Staubli VAL3: POLYGON.dtx

public num distance
public num moveType = 1
public num nIndexGun
public num nStop
public num nTcpAction = 1
public num nTime
public num nEdge
public num nRotationangle
public num nWidth
public num nLaserDelay = 0.8
public num nLaserPower = 60
public num nGasPressure = 90
public num nFrameIndex
public num nPWMPercent = 100
public num nJointMode
public string comment = "Polygon..."
public string instruction
public bool bCutting
public bool toStop
public bool bRes
public frame fTrack = {fatherId=world[0]}
public jointRx jReadyInOut
public jointRx jConfig
public pointRx pMoveTo = {fatherId=fTrack[0]}
public pointRx pCutting[21]
  [0] = {fatherId=fTrack[0]}
  [1] = {fatherId=fTrack[0]}
  [2] = {fatherId=fTrack[0]}
  [3] = {fatherId=fTrack[0]}
  [4] = {fatherId=fTrack[0]}
  [5] = {fatherId=fTrack[0]}
  [6] = {fatherId=fTrack[0]}
  [7] = {fatherId=fTrack[0]}
  [8] = {fatherId=fTrack[0]}
  [9] = {fatherId=fTrack[0]}
  [10] = {fatherId=fTrack[0]}
  [11] = {fatherId=fTrack[0]}
  [12] = {fatherId=fTrack[0]}
  [13] = {fatherId=fTrack[0]}
  [14] = {fatherId=fTrack[0]}
  [15] = {fatherId=fTrack[0]}
  [16] = {fatherId=fTrack[0]}
  [17] = {fatherId=fTrack[0]}
  [18] = {fatherId=fTrack[0]}
  [19] = {fatherId=fTrack[0]}
  [20] = {fatherId=fTrack[0]}
public pointRx pFirst = {fatherId=fTrack[0]}
public pointRx pSecond = {fatherId=fTrack[0]}
public pointRx pThird = {fatherId=fTrack[0]}
public pointRx points = {fatherId=fTrack[0]}
public pointRx pO = {fatherId=world[0]}
public pointRx pX = {fatherId=world[0]}
public pointRx pY = {fatherId=world[0]}
public mdesc nom_speed = {accel=3.333333, vel=33.333333, decel=3.333333, tmax=66.666667, rmax=60, leave=0.05, reach=0.05, blend=off}
public mdesc mJointSpeed = {vel=50, tmax=9999, rmax=9999, leave=30, reach=30}
